INTERFACE ITF_BaseGroupElement_HMI_Connector_Command

END_INTERFACE

(* stored: Version 1.1.0.1
   Itf ITF_BaseGroupElement_HMI_Connector_Command: Id {af9c5ec1-f410-0848-0c82-380e31ef43f2} *)
